FUNCTION Convert_ULINT_TO_DT : BOOL
VAR_INPUT
	in : ULINT;
	out : REFERENCE TO DT;
END_VAR
VAR
	converted : DT;
END_VAR

converted := ULINT_TO_DT(in);

IF (DT_TO_ULINT(converted) <> in) THEN
	RETURN;
END_IF

out := converted;
Convert_ULINT_TO_DT := TRUE;

END_FUNCTION

(* stored: Version 1.1.0.1, ProductVersion 3.1.4024.12
   POU Convert_ULINT_TO_DT: Id {a357d4a1-562d-4ce0-acc2-f07556205db6}, SpecialFunc None *)
